// TwinCAT 3 PLC project Test
// ProgramVersion: 3.1.0.8
// libraries:
//   FloatingPointUtils, * (System)
//   Tc2_ModbusSrv, * (Beckhoff Automation GmbH)
//   Tc2_Standard, * (Beckhoff Automation GmbH)
//   Tc2_System, * (Beckhoff Automation GmbH)
//   Tc2_Utilities, * (Beckhoff Automation GmbH)
//   Tc3_Interfaces, * (Beckhoff Automation GmbH)
//   Tc3_Module, * (Beckhoff Automation GmbH)
// project tree:
//   GVLs/ GVL.TcGVL
//   / PlcTask.TcTTO (not stored)
//   POUs/ FB_ModbusPoll.TcPOU, MAIN.TcPOU

// ---- GVLs/GVL.TcGVL
VAR_GLOBAL
	arr AT%MW0: ARRAY [0..2] OF WORD;
END_VAR

// ---- POUs/FB_ModbusPoll.TcPOU
FUNCTION_BLOCK FB_ModbusPoll

VAR_INPUT
	ipAd : STRING; // the ip address of the modbus server
	startAddr : WORD; // the start address
END_VAR

VAR_OUTPUT
	dataStr : STRING;
END_VAR

VAR
	bModbusTick : BOOL;
	fbReadRegs : FB_MBReadInputRegs;
END_VAR

fbReadRegs.sIPAddr := ipAd; //gateway ip
fbReadRegs.nTCPPort := MODBUS_TCP_PORT; //502
fbReadRegs.nUnitID := 16#FF; //255
fbReadRegs.nQuantity := 3; //3 words
fbReadRegs.tTimeout := T#5S; //30 sec timout
fbReadRegs.nMBAddr := startAddr;
fbReadRegs.cbLength := 6;//nq*2
fbReadRegs.pDestAddr := ADR(arr); //the pointer to the array

//the rising edge of the input negate the tick to create  a rising input of change :)
fbReadRegs.bExecute := (bModbusTick := NOT bModbusTick); 

//uppercase(convert first number to hex + convert second number to hex)
dataStr := F_TOUCase(CONCAT(WORD_TO_HEXSTR(arr[1],4,TRUE),WORD_TO_HEXSTR(arr[2],4,TRUE))); 
fbReadRegs();

END_FUNCTION_BLOCK

// ---- POUs/MAIN.TcPOU
PROGRAM MAIN
VAR
str : STRING;
poll : FB_ModbusPoll;
actualData AT%MW0: REAL;
t:REAL;
END_VAR


poll.ipAd := '192.168.1.101';
poll.startAddr := 0;
poll(dataStr => str);
FPU.HexStrToReal(str := CONCAT('16#',str), f => t);
FPU.HexStrToReal(str:=str , f=> t)

END_PROGRAM
